(* CoDeSys 2.3.10.0 project: Servo.pro *)
(* Libraries: STANDARD.LIB 5.6.98 12:03:02 *)

(* Task configuration *)
TASK Standard (PRIORITY := 0, INTERVAL := T#10ms);
	MAIN();
END_TASK

(* Global variable list: Global_Variables *)
VAR_GLOBAL
	Zielona_1 		AT 	%Q* 	:	 BOOL:= 0;
	Zielona_2 		AT 	%Q* 	:	 BOOL:= 0;
	Zielona_3 		AT 	%Q* 	:	 BOOL:= 0;
	Zielona_4 		AT 	%Q* 	:	 BOOL:= 0;

	Czerwona_1 		AT 	%Q*		:	 BOOL:= 0;
	Czerwona_2 		AT 	%Q*		:	 BOOL:= 0;
	Czerwona_3 		AT	%Q*		:	 BOOL:= 0;
	Czerwona_4 		AT 	%Q*		:	 BOOL:= 0;

	Przycisk_1 		AT 	%I*		:	BOOL;
	Przycisk_2 		AT 	%I*		: 	BOOL;
	Przycisk_3 		AT 	%I*		: 	BOOL;
	Przycisk_4 		AT 	%I*		: 	BOOL;

	RegulatorIn_1 	AT 	%I*		:	INT;
	RegulatorIn_2 	AT 	%I*		:	INT;

	RegulatorOut_1 	AT 	%Q*		:	UDINT;
	RegulatorOut_2 	AT 	%Q*		:	UDINT;

	Scale_1			AT	%Q*		:	INT;
	Scale_2			AT	%Q*		:	INT;

	Enable_1		AT	%Q*		:	BOOL;
	Enable_2		AT 	%Q*		:	BOOL;

	axis1_Not_moving		AT 	%I*		:	BOOL;
	axis1_Moving_Fv		AT 	%I*		:	BOOL;
	axis1_Moving_Bw		AT 	%I*		:	BOOL;
	axis1_position		AT 	%I*		:	LREAL;

	axis2_Not_moving		AT 	%I*		:	BOOL;
	axis2_Moving_Fv		AT 	%I*		:	BOOL;
	axis2_Moving_Bw		AT 	%I*		:	BOOL;
	axis2_position		AT 	%I*		:	LREAL;

	state_device1		AT 	%I*		:	UINT;
	state_device2		AT 	%I*		:	UINT;
	state_device3		AT 	%I*		:	UINT;
	state_device4		AT 	%I*		:	UINT;
	state_device5		AT 	%I*		:	UINT;
	state_device6		AT 	%I*		:	UINT;
	state_device7		AT 	%I*		:	UINT;
	state_device8		AT 	%I*		:	UINT;
(*	Velo_1			AT	%I*		:	LREAL;*)
(*	Velo_2			AT	%I*		:	LREAL;*)
END_VAR

(* Global variable list: TwinCAT_Configuration *)
(* Generated automatically by TwinCAT - (read only) *)
VAR_CONFIG
	.Zielona_1 AT %QX0.0 : BOOL;
	.Zielona_2 AT %QX0.1 : BOOL;
	.Zielona_3 AT %QX0.2 : BOOL;
	.Zielona_4 AT %QX0.3 : BOOL;
	.Czerwona_1 AT %QX0.4 : BOOL;
	.Czerwona_2 AT %QX0.5 : BOOL;
	.Czerwona_3 AT %QX0.6 : BOOL;
	.Czerwona_4 AT %QX0.7 : BOOL;
	.Przycisk_1 AT %IX0.0 : BOOL;	(*  ~ {LinkedWith:TIID^Device 2 (EtherCAT (v2.10 only))^Term 3 (EK1100)^Przyciski (EL1004)^Channel 1^Input} *)
	.Przycisk_2 AT %IX0.1 : BOOL;	(*  ~ {LinkedWith:TIID^Device 2 (EtherCAT (v2.10 only))^Term 3 (EK1100)^Przyciski (EL1004)^Channel 2^Input} *)
	.Przycisk_3 AT %IX0.2 : BOOL;	(*  ~ {LinkedWith:TIID^Device 2 (EtherCAT (v2.10 only))^Term 3 (EK1100)^Przyciski (EL1004)^Channel 3^Input} *)
	.Przycisk_4 AT %IX0.3 : BOOL;	(*  ~ {LinkedWith:TIID^Device 2 (EtherCAT (v2.10 only))^Term 3 (EK1100)^Przyciski (EL1004)^Channel 4^Input} *)
	.RegulatorIn_1 AT %IB4 : INT;
	.RegulatorIn_2 AT %IB6 : INT;
	.RegulatorOut_1 AT %QB4 : UDINT;
	.RegulatorOut_2 AT %QB8 : UDINT;
	.Scale_1 AT %QB12 : INT;
	.Scale_2 AT %QB14 : INT;
	.Enable_1 AT %QX16.0 : BOOL;
	.Enable_2 AT %QX16.1 : BOOL;
	.axis1_Not_moving AT %IX8.0 : BOOL;	(*  ~ {LinkedWith:TINC^NC-Task 1 SAF^Axes^Axis 1^Outputs^Axis 1_ToPlc^StateDWord^NotMoving} *)
	.axis1_Moving_Fv AT %IX8.1 : BOOL;	(*  ~ {LinkedWith:TINC^NC-Task 1 SAF^Axes^Axis 1^Outputs^Axis 1_ToPlc^StateDWord^PositiveDirection} *)
	.axis1_Moving_Bw AT %IX8.2 : BOOL;	(*  ~ {LinkedWith:TINC^NC-Task 1 SAF^Axes^Axis 1^Outputs^Axis 1_ToPlc^StateDWord^NegativeDirection} *)
	.axis1_position AT %IB44 : LREAL;	(*  ~ {LinkedWith:TINC^NC-Task 1 SAF^Axes^Axis 1^Outputs^Axis 1_ToPlc^ActPos} *)
	.axis2_Not_moving AT %IX8.3 : BOOL;	(*  ~ {LinkedWith:TINC^NC-Task 1 SAF^Axes^Axis 2^Outputs^Axis 2_ToPlc^StateDWord^NotMoving} *)
	.axis2_Moving_Fv AT %IX8.4 : BOOL;	(*  ~ {LinkedWith:TINC^NC-Task 1 SAF^Axes^Axis 2^Outputs^Axis 2_ToPlc^StateDWord^PositiveDirection} *)
	.axis2_Moving_Bw AT %IX8.5 : BOOL;	(*  ~ {LinkedWith:TINC^NC-Task 1 SAF^Axes^Axis 2^Outputs^Axis 2_ToPlc^StateDWord^NegativeDirection} *)
	.axis2_position AT %IB34 : LREAL;	(*  ~ {LinkedWith:TINC^NC-Task 1 SAF^Axes^Axis 2^Outputs^Axis 2_ToPlc^ActPos} *)
	.state_device1 AT %IB12 : UINT;	(*  ~ {LinkedWith:TIID^Device 2 (EtherCAT (v2.10 only))^Drive 1 (AX5203-0000-0010)^InfoData^State} *)
	.state_device2 AT %IB16 : UINT;	(*  ~ {LinkedWith:TIID^Device 2 (EtherCAT (v2.10 only))^Term 3 (EK1100)^InfoData^State} *)
	.state_device3 AT %IB18 : UINT;	(*  ~ {LinkedWith:TIID^Device 2 (EtherCAT (v2.10 only))^Term 3 (EK1100)^Term 4 (EL4132)^InfoData^State} *)
	.state_device4 AT %IB20 : UINT;	(*  ~ {LinkedWith:TIID^Device 2 (EtherCAT (v2.10 only))^Term 3 (EK1100)^Zielone (EL2004)^InfoData^State} *)
	.state_device5 AT %IB22 : UINT;	(*  ~ {LinkedWith:TIID^Device 2 (EtherCAT (v2.10 only))^Term 3 (EK1100)^Przyciski (EL1004)^InfoData^State} *)
	.state_device6 AT %IB24 : UINT;	(*  ~ {LinkedWith:TIID^Device 2 (EtherCAT (v2.10 only))^Term 3 (EK1100)^Czerwone (EL2004)^InfoData^State} *)
	.state_device7 AT %IB26 : UINT;	(*  ~ {LinkedWith:TIID^Device 2 (EtherCAT (v2.10 only))^Term 3 (EK1100)^Term 8 (EL3102)^InfoData^State} *)
	.state_device8 AT %IB28 : UINT;
END_VAR

(* POU MAIN, ST *)
PROGRAM MAIN
VAR
	test: UINT := 100;
	stoper_device1: STOPWATCH := (max_value:=t#20s);
	stoper_device2: STOPWATCH := (max_value:=t#20s);
	stoper_device3: STOPWATCH := (max_value:=t#20s);
	stoper_device4: STOPWATCH := (max_value:=t#20s);
	stoper_device5: STOPWATCH := (max_value:=t#20s);
	stoper_device6: STOPWATCH := (max_value:=t#20s);
	stoper_device7: STOPWATCH := (max_value:=t#20s);
	stoper_device8: STOPWATCH := (max_value:=t#20s);

	stoper_axis1: STOPWATCH := (max_value:=t#120s);
	stoper_axis2: STOPWATCH := (max_value:=t#120s);
END_VAR
Czerwona_1 :=  NOT Przycisk_1;
Czerwona_2 :=  NOT Przycisk_2;
Czerwona_3 :=  NOT Przycisk_3;
Czerwona_4 :=  NOT Przycisk_4;

Zielona_1:=  Przycisk_1;
Zielona_2:=  Przycisk_2;
Zielona_3:=  Przycisk_3;
Zielona_4:=  Przycisk_4;

Enable_1 := TRUE;
Enable_2 := TRUE;

Scale_1 := 100;
Scale_2 := 100;
test := 100;

stoper_device1.start_stop := state_device1 <> 8;
stoper_device1();
stoper_device2.start_stop := state_device2 <> 8;
stoper_device2();
stoper_device3.start_stop := state_device3 <> 8;
stoper_device3();
stoper_device4.start_stop := state_device4 <> 8;
stoper_device4();
stoper_device5.start_stop := state_device5 <> 8;
stoper_device5();
stoper_device6.start_stop := state_device6 <> 8;
stoper_device6();
stoper_device7.start_stop := state_device7 <> 8;
stoper_device7();
stoper_device8.start_stop := state_device8 <> 8;
stoper_device8();

stoper_axis1.start_stop := NOT axis1_Not_moving;
stoper_axis1();
stoper_axis2.start_stop := NOT axis2_Not_moving;
stoper_axis2();


IF (RegulatorIn_1   < 100) AND (RegulatorIn_1   > 0) THEN
	RegulatorOut_1 := RegulatorIn_1 * 10000;
ELSE IF (RegulatorIn_1   > 100) THEN
		RegulatorOut_1 := 100 * 10000;
END_IF;
END_IF;

IF (RegulatorIn_2   < 100) AND (RegulatorIn_2   > 0) THEN
	RegulatorOut_2 := RegulatorIn_2 * 10000;
ELSE IF (RegulatorIn_2   > 100) THEN
		RegulatorOut_2 := 100 * 10000;
END_IF;
END_IF;
END_PROGRAM

(* POU STOPWATCH, ST *)
FUNCTION_BLOCK STOPWATCH
VAR_INPUT
	max_value: TIME:=t#10S;
	start_stop: BOOL := FALSE;
END_VAR
VAR_OUTPUT
	value: TIME := t#0s;
END_VAR
VAR
	timer: TON;
END_VAR
IF timer.PT <> max_value THEN
	timer.PT := max_value;
END_IF;

IF start_stop = TRUE THEN
	timer(IN:=TRUE);
	value :=timer.ET;
ELSE
	IF timer.IN THEN
		value :=timer.ET;
	END_IF;
	timer(IN:=FALSE);
END_IF;
END_FUNCTION_BLOCK

(* Visualisation StandState
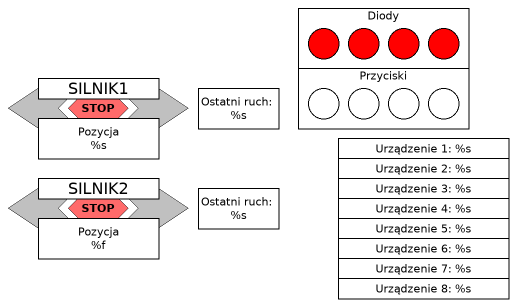
rounded rectangle at (320,0)-(491,61): text "Diody"
polygon at (150,80)-(210,120): invisible if NOT axis1_Moving_Fv
polygon at (30,80)-(90,120): invisible if NOT axis1_Moving_Bw
polygon at (90,90)-(150,110): text "STOP"; invisible if NOT axis1_Not_moving
ellipse at (330,20)-(361,51): invisible if NOT Zielona_1
polygon at (150,180)-(210,220): invisible if NOT axis2_Moving_Fv
polygon at (30,180)-(90,220): invisible if NOT axis2_Moving_Bw
polygon at (90,190)-(150,210): text "STOP"; invisible if NOT axis2_Not_moving
ellipse at (330,20)-(361,51): invisible if NOT Czerwona_1
rectangle at (360,130)-(531,151): text "Urządzenie 1: %s"; shows MAIN.stoper_device1.value
rectangle at (220,80)-(301,121): text "Ostatni ruch: / %s"; shows MAIN.stoper_axis1.value
rectangle at (220,180)-(301,221): text "Ostatni ruch: / %s"; shows MAIN.stoper_axis2.value
ellipse at (370,20)-(401,51): invisible if NOT Zielona_2
ellipse at (370,20)-(401,51): invisible if NOT Czerwona_2
ellipse at (410,20)-(441,51): invisible if NOT Zielona_3
ellipse at (410,20)-(441,51): invisible if NOT Czerwona_3
ellipse at (450,20)-(481,51): invisible if NOT Zielona_4
ellipse at (450,20)-(481,51): invisible if NOT Czerwona_4
rectangle at (360,150)-(531,171): text "Urządzenie 2: %s"; shows MAIN.stoper_device2.value
rectangle at (360,170)-(531,191): text "Urządzenie 3: %s"; shows MAIN.stoper_device3.value
rectangle at (360,190)-(531,211): text "Urządzenie 4: %s"; shows MAIN.stoper_device4.value
rectangle at (360,210)-(531,231): text "Urządzenie 5: %s"; shows MAIN.stoper_device5.value
rectangle at (360,230)-(531,251): text "Urządzenie 6: %s"; shows MAIN.stoper_device6.value
rectangle at (360,250)-(531,271): text "Urządzenie 7: %s"; shows MAIN.stoper_device7.value
rectangle at (360,270)-(531,291): text "Urządzenie 8: %s"; shows MAIN.stoper_device8.value
rectangle at (60,70)-(181,91): text "SILNIK1"
rectangle at (60,170)-(181,191): text "SILNIK2"
rounded rectangle at (320,60)-(491,121): text "Przyciski"
ellipse at (330,80)-(361,111): alarm colour if Przycisk_1
ellipse at (370,80)-(401,111): alarm colour if Przycisk_2
ellipse at (410,80)-(441,111): alarm colour if Przycisk_3
ellipse at (450,80)-(481,111): alarm colour if Przycisk_4
rectangle at (60,110)-(181,151): text "Pozycja / %s"; shows axis1_position
rectangle at (60,210)-(181,251): text "Pozycja / %f"; shows axis2_position
*)
